FUNCTION_BLOCK TcoHardwareDiagContext EXTENDS TcoCore.TcoContext
VAR
	_BackPlane : EthercatMasterBase(THIS^);
	_X001 : EthercatMasterAdditionalSyncUnit(THIS^);
END_VAR

METHOD PROTECTED MAIN
VAR_INPUT
END_VAR
_BackPlane.Diagnostics();
_X001.Diagnostics();
END_METHOD

END_FUNCTION_BLOCK

(* stored: Version 1.1.0.1, ProductVersion 3.1.4024.9
   POU TcoHardwareDiagContext: Id {e2f5ead5-24ed-0ea9-1b23-b0fd0d86ba2f}, SpecialFunc None
   Method MAIN: Id {e941468e-7823-08cb-1726-ee54f1441bb1} *)
